INTERFACE I_Logger

END_INTERFACE

(* stored: Version 1.1.0.1
   Itf I_Logger: Id {8d10f800-b621-4e55-9c3b-f2a551bf051a} *)
